(* CODESYS project Flight Simulator Diagnostics.project.export

Project tree, tasks and I/O mapping:
  application Application
    libraries: Unit Conversion Interfaces, * (Intern); Standard, * (System); VisuDialogs, * (System); CAA Device Diagnosis, 3.5.4.0 (CAA Technical Workgroup); CAA Net Base Services, 3.5.8.10 (CAA Technical Workgroup); NetVarUdp, 3.5.17.0 (System); PRO JSON, 1.0.0.13 (Pro Electric)
    task EtherCAT_Task (cyclic, interval 8 ms, priority 1) calls nothing
    task VISU_TASK (cyclic, interval 200 ms, priority 31) calls VisuElems.Visu_Prg
    task Task (cyclic, interval 5 ms, priority 1) calls main, TcpClient
    global variables gvlSetting
    data type ServoData
    program TcpClient [ST]
    program main [ST]
    visualisation Main
    global variables GVL
    program DriveDiagnostics [ST]
    function AppendDiagnosticText [ST]
    function BuildDiagnosticFeedback [ST]
*)

// Application/ServoData
TYPE ServoData :
STRUCT
	positions: ARRAY[1..6] OF JSONVAR;
	speeds: ARRAY[1..6] OF JSONVAR;
END_STRUCT
END_TYPE

// Application/gvlSetting
{attribute 'qualified_only'}
VAR_GLOBAL CONSTANT
    // Port to use to send data.
	gc_uiPort        : UINT := 32760;
    // IP Address of the computer that hosts the software.
	gc_stIpAddr      : NBS.IP_ADDR := (sAddr := '192.168.137.123');
	// Length of the telegram.
    gc_wMaxTelegram  : INT := 512;
END_VAR

// Application/GVL
{attribute 'qualified_only'}
VAR_GLOBAL
	// Red light on electrical housing.
	lightRed: BOOL;
	// Yellow light on electrical housing.
	lightYellow: BOOL;
	// Green light on electrical housing.
	lightGreen: BOOL;
	// Reset button on electrical housing.
	resetButton: BOOL := FALSE;
	// Start button on electrical housing.
	startButton: BOOL := FALSE;
	// Stop button on electrical housing.
	stopButton: BOOL := FALSE;
	// Safety system, connected to safety relay.
	safetySystem: BOOL := FALSE;
	// Virtual reset button on HMI.
	resetHMI: BOOL;
	// Virtual start button on HMI.
	startHMI: BOOL;
	// Virtual stop button on HMI.
	stopHMI: BOOL;
	// Virtual toggle button to toggle between tCP data and manual data on HMI.
	useTCPData: BOOL := TRUE;
	// Manual slider velocity input on HMI.
	nextVelocityInput: REAL := 200;
	// Manual slider position input on HMI.
	nextPositionInput: REAL := 0;
	// Flight simulator object.
	FlightSimulator: FlightSimulator;
	// Velocity input from TCP data or HMI data.
	servoVelocities: ARRAY[1..6] OF REAL;
	// Position input from TCP data or HMI data.
	servoPositions: ARRAY[1..6] OF REAL;
	// Current Positions in array format.
	servoPositionsCurrent: ARRAY[1..6] OF REAL;
	// Current Positions in JSON format, used to send back to TCP client.
	currentPositions: ARRAY[1..6] OF JSONVAR;
END_VAR

// Application/main
PROGRAM main
VAR
	bInit: BOOL := TRUE;
	iCounter : INT;
	bEnabled: BOOL;
	iDataUpdated: INT := 0;
	tonTimer: TON;
	UpdateCount: INT := 0;
END_VAR

IF bInit THEN
	GVL.FlightSimulator.init(
		axis1 := servo_drive_1,
		axis2 := servo_drive_2,
		axis3 := servo_drive_3,
		axis4 := servo_drive_4,
		axis5 := servo_drive_5,
		axis6 := servo_drive_6,
		GVL.lightRed,
		GVL.lightYellow,
		GVL.lightGreen,
		enabled := bEnabled,
		safetySystem := GVL.safetySystem,
		newPositions := GVL.servoPositions,
		newVelocities := GVL.servoVelocities
	);
	bInit := FALSE;
END_IF

// Handle reset buttons.
IF GVL.resetButton OR GVL.resetHMI THEN // blauwe knop
	bEnabled := FALSE;
	GVL.FlightSimulator.doReset();
	
	// [NEW] Reset position data zodat platform niet naar oude waarden springt
	FOR iCounter := 1 TO 6 DO
		GVL.currentPositions[iCounter].Number := 0.0;
		GVL.servoPositions[iCounter] := 0.0;
		GVL.servoVelocities[iCounter] := 0.0;
	END_FOR
END_IF

// Handle start buttons.
IF GVL.startButton OR GVL.startHMI THEN // witte knop
	bEnabled := TRUE;
END_IF

// Handle stop buttons
IF GVL.stopButton OR GVL.stopHMI THEN // zwarte knop
	bEnabled := FALSE;
END_IF

// Go through all positions and velocities.
FOR iCounter := 1 TO 6 BY 1 DO 
	IF GVL.useTCPData THEN
		// Always use latest TCP data (don't wait for parseJSON.Done)
		GVL.servoPositions[iCounter] := tcpClient.servoData.positions[iCounter].Number;
		GVL.servoVelocities[iCounter] := tcpClient.servoData.speeds[iCounter].Number;
		
		// Optional: track successful updates for diagnostics
		IF tcpClient.parseJSON.Done THEN
			UpdateCount := UpdateCount + 1;
		END_IF
	ELSE
		// Else take the data from the sliders from the HMI.
		GVL.servoPositions[iCounter] := GVL.nextPositionInput;
		GVL.servoVelocities[iCounter] := GVL.nextVelocityInput;
	END_IF
END_FOR

//THIS^.signal.green.enable := FALSE;
//THIS^.signal.green.blink := FALSE;
//THIS^.signal.green.enable := FALSE;
//THIS^.signal.green.blink := FALSE;

// Cycle sub functions.
GVL.FlightSimulator.cycle();

// Get current positions, used for TcpClient.
FOR iCounter := 1 TO 6 BY 1 DO
	GVL.currentPositions[iCounter].Number := GVL.FlightSimulator.axis[iCounter].getPosition();
	GVL.servoPositionsCurrent[iCounter] := GVL.FlightSimulator.axis[iCounter].getPosition();
END_FOR

END_PROGRAM

// Application/TcpClient
PROGRAM TcpClient
VAR

    // Client object that connects to client machine.
	fbTcpClient   : NBS.TCP_Client;
    // Read object that reads incomming data from client machine.
	fbTcpRead     : NBS.TCP_Read;
    // Write object that writes data to client machine.
	fbTcpWrite    : NBS.TCP_Write;
	
	// TON object for reset delay.
	tonResetDelay: TON;
	// Received telegram from Read object.
	received      : STRING(gvlSetting.gc_wMaxTelegram);
	// Sent telegram to Write object.
	sent          : STRING(4095);
	// JSON Parser object to parse read data.
	parseJSON     : JSON_TO_STRUCT;
	// JSON Composer object to compose data to write.
	composeJSON   : STRUCT_TO_JSON;
	// Struct that stores the received data in usable arrays.
	servoData     : ServoData;
    // Make connection.
	xConnect      : BOOL := TRUE;
	// Do composing.
	xCompose: BOOL;
	// Do write action.
	xWrite: BOOL;
	// Do parsing
	xParse: BOOL;
	
	j : INT := 1;
 
    // Do read action.
	xRead         : BOOL;
    // Size of read data telegram.
	udiRead       : UDINT;
	// Timeout in µs.
	udiTimeOut: UDINT := 500000;
	
	
	udiVal        : UDINT;
    pudiVal       : POINTER TO BYTE;
    iIndex        : INT;
	xMissingAck   : BOOL;
    udiResult     : UDINT;
    udiLastAck    : UDINT;
    udiNow        : UDINT;
    diagnosticSendTimer : TON;
    diagnosticBuildErrors : UDINT;
END_VAR

 fbTcpClient(xEnable := xConnect, ipAddr := gvlSetting.gc_stIpAddr, uiPort := gvlSetting.gc_uiPort, udiTimeOut := udiTimeOut);
// 
// // Run when connection is active.
// IF fbTcpClient.xActive AND GVL.FlightSimulator.isInitialised() THEN
// 	
// 	IF fbTcpWrite.xDone THEN
// 		xWrite := FALSE;
// 	ELSIF NOT fbTcpWrite.xBusy THEN
// 		IF composeJSON.Done AND composeJSON.Execute THEN
// 			xCompose := FALSE;
// 			xWrite := TRUE;
// 		ELSIF (NOT composeJSON.Busy) THEN
// 			   xCompose := TRUE;
// 			   xWrite := FALSE;
// 		END_IF
// 	END_IF
// 	
// 	composeJSON(
// 		Execute:= xCompose,
// 		JSONString:= ADR(sent),
// 		JSONStringSize:= SIZEOF(sent),
// 		JSONVars:= ADR(GVL.currentPositions),
// 		NumberOfVars:= SIZEOF(GVL.currentPositions) / SIZEOF(JSONVAR)
// 	); 
// 	fbTcpWrite(xExecute := xWrite, hConnection := fbTcpClient.hConnection, udiTimeOut := udiTimeOut, szSize := SIZEOF(sent), pData := ADR(sent));
// 	
// 	IF (NOT fbTcpRead.xBusy) AND (NOT parseJSON.Busy) THEN
// 		xRead := TRUE;
// 	ELSIF fbTcpRead.xReady THEN
// 		xRead := FALSE;
// 		xParse := TRUE;
// 	ELSIF (NOT parseJSON.Busy) THEN
// 		xParse := FALSE;
// 	END_IF
// 
// 	parseJSON(
// 		Execute := xParse,
// 		JSONString:= ADR(received),
// 		JSONStringSize:= SIZEOF(received),
// 		JSONVars:= ADR(servoData),
// 		NumberOfVars:= SIZEOF(servoData) / SIZEOF(JSONVAR)
// 	);
// 	
// 	received := '';
// 	//FOR j := 1 TO SIZEOF(received) DO
// 	//	received[j] := 0;
// 	//END_FOR
// 	//sent := '';
// 	fbTcpRead(xEnable := xRead, hConnection := fbTcpClient.hConnection, szSize := SIZEOF(received), pData := ADR(received), szCount => udiRead);
// 	
// END_IF
// 
// // Reset connection when connection has stopped.
// IF (NOT xConnect) THEN
// 	// Reset all variables.
// 	xConnect := FALSE;
// 	xWrite := FALSE;
// 	xCompose := FALSE;
// 	fbTcpWrite(xExecute := FALSE);
// 	xRead := FALSE;
// 	xParse := FALSE;
// 	fbTcpRead(xEnable := FALSE);
// 	received := '';
// 	sent := '';
// 	// Delay reset for 3 sec.
// 	tonResetDelay(IN:=TRUE, PT:=T#3S);
// 	IF (tonResetDelay.Q) THEN
// 		tonResetDelay(IN:=FALSE);
// 		xConnect := TRUE;
// 	END_IF
// 	
// END_IF
// 
// IF fbTcpClient.xDone AND xConnect THEN
// 	xConnect := FALSE;
// END_IF
// 
// // Stop connection when in error.
// //IF fbTcpClient.xError OR fbTcpWrite.xError OR fbTcpRead.xError THEN
// IF fbTcpClient.xError OR fbTcpRead.xError THEN
// 
// 	xConnect := FALSE;
// 	fbTcpWrite(xExecute := FALSE);
// END_IF 
// 

// Run when connection is active.
IF fbTcpClient.xActive AND GVL.FlightSimulator.isInitialised() THEN
    DriveDiagnostics();
    diagnosticSendTimer(IN := NOT xWrite, PT := T#50MS);
    IF fbTcpWrite.xDone OR fbTcpWrite.xError THEN
        xWrite := FALSE;
    ELSIF NOT fbTcpWrite.xBusy AND diagnosticSendTimer.Q THEN
        sent := BuildDiagnosticFeedback();
        xWrite := LEN(sent) > 0;
        IF NOT xWrite THEN diagnosticBuildErrors := diagnosticBuildErrors + 1; END_IF
    END_IF
    // Buffer remains unchanged while TCP_Write is busy. Send only meaningful
    // bytes (including the newline), never the unused NUL-filled capacity.
    fbTcpWrite(xExecute := xWrite, hConnection := fbTcpClient.hConnection,
        udiTimeOut := udiTimeOut, szSize := INT_TO_UDINT(LEN(sent)), pData := ADR(sent));

    // -------------------------
    //  ONTVANGEN VAN STUARTSERVER
    // -------------------------
    IF (NOT fbTcpRead.xBusy) AND (NOT parseJSON.Busy) THEN
        xRead := TRUE;
    ELSIF fbTcpRead.xReady THEN
        xRead := FALSE;
        xParse := TRUE;
    ELSIF (NOT parseJSON.Busy) THEN
        xParse := FALSE;
    END_IF

    parseJSON(
        Execute         := xParse,
        JSONString      := ADR(received),
        JSONStringSize  := SIZEOF(received),
        JSONVars        := ADR(servoData),
        NumberOfVars    := SIZEOF(servoData) / SIZEOF(JSONVAR)
    );

    // Buffer leegmaken voor volgende receive
    received := '';
    fbTcpRead(
        xEnable    := xRead,
        hConnection:= fbTcpClient.hConnection,
        szSize     := SIZEOF(received),
        pData      := ADR(received),
        szCount    => udiRead
    );

END_IF


// Reset connection when connection has stopped.
 IF (NOT xConnect) THEN
 	// Reset all variables.
 	xConnect := FALSE;
 	xWrite := FALSE;
 	xCompose := FALSE;
	fbTcpWrite(xExecute := FALSE);
 	xRead := FALSE;
 	xParse := FALSE;
 	fbTcpRead(xEnable := FALSE);
	received := '';
 	sent := '';
 	// Delay reset for 3 sec.
 	tonResetDelay(IN:=TRUE, PT:=T#3S);
 	IF (tonResetDelay.Q) THEN
 		tonResetDelay(IN:=FALSE);
 		xConnect := TRUE;
 	END_IF
	
 END_IF
 
 IF fbTcpClient.xDone AND xConnect THEN
 	xConnect := FALSE;
 END_IF

 // Stop connection when in error.
 //IF fbTcpClient.xError OR fbTcpWrite.xError OR fbTcpRead.xError THEN
IF fbTcpClient.xError OR fbTcpRead.xError THEN

	xConnect := FALSE;
	fbTcpWrite(xExecute := FALSE);
END_IF

END_PROGRAM

// Application/DriveDiagnostics
PROGRAM DriveDiagnostics
VAR
    // Passive readers only. No command, enable, reset, or axis configuration writes.
    positionReaders : ARRAY[1..6] OF MC_ReadActualPosition_Festo;
    velocityReaders : ARRAY[1..6] OF MC_ReadActualVelocity_Festo;
    parameterReader : MC_ReadParameter_Festo;
    actualPositions : ARRAY[1..6] OF REAL;
    actualVelocities : ARRAY[1..6] OF REAL;
    positionValid : ARRAY[1..6] OF BOOL;
    velocityValid : ARRAY[1..6] OF BOOL;
    driveTargets : ARRAY[1..6] OF LREAL;
    followingErrors : ARRAY[1..6] OF LREAL;
    targetNew : ARRAY[1..6] OF BOOL;
    followingNew : ARRAY[1..6] OF BOOL;
    targetTick : ARRAY[1..6] OF UDINT;
    followingTick : ARRAY[1..6] OF UDINT;
    readErrors : ARRAY[1..6] OF WORD;
    readErrorCount : UDINT;
    sampleSequence : UDINT;
    sampleTick : UDINT;
    pollAxis : INT := 1;
    pollFollowing : BOOL;
    pollActive : BOOL;
    pollReset : BOOL;
    pollInterval : TON;
    pollTimeout : TON;
    parameter : UINT;
    drive : REFERENCE TO AXIS_REF_FESTO;
    i : INT;
END_VAR

// User units are supplied by the Festo library. Valid AND NOT Error is required;
// never turn a failed read into a plausible zero-valued measurement.
positionReaders[1](Axis := servo_drive_1, Enable := TRUE);
positionReaders[2](Axis := servo_drive_2, Enable := TRUE);
positionReaders[3](Axis := servo_drive_3, Enable := TRUE);
positionReaders[4](Axis := servo_drive_4, Enable := TRUE);
positionReaders[5](Axis := servo_drive_5, Enable := TRUE);
positionReaders[6](Axis := servo_drive_6, Enable := TRUE);
velocityReaders[1](Axis := servo_drive_1, Enable := TRUE);
velocityReaders[2](Axis := servo_drive_2, Enable := TRUE);
velocityReaders[3](Axis := servo_drive_3, Enable := TRUE);
velocityReaders[4](Axis := servo_drive_4, Enable := TRUE);
velocityReaders[5](Axis := servo_drive_5, Enable := TRUE);
velocityReaders[6](Axis := servo_drive_6, Enable := TRUE);
sampleTick := TIME_TO_UDINT(TIME());
FOR i := 1 TO 6 DO
    positionValid[i] := positionReaders[i].Valid AND NOT positionReaders[i].Error;
    velocityValid[i] := velocityReaders[i].Valid AND NOT velocityReaders[i].Error;
    actualPositions[i] := positionReaders[i].Position;
    actualVelocities[i] := velocityReaders[i].Velocity;
END_FOR

// Only one SDO request is active across all six drives. Each request is followed
// by a 50 ms idle interval. Register traces are slower than the 20 Hz PDO traces.
// Do not increase this rate without measuring the actual fieldbus load.
CASE pollAxis OF
    1: drive REF= servo_drive_1;
    2: drive REF= servo_drive_2;
    3: drive REF= servo_drive_3;
    4: drive REF= servo_drive_4;
    5: drive REF= servo_drive_5;
    6: drive REF= servo_drive_6;
END_CASE
IF pollFollowing THEN parameter := 16#60F4; ELSE parameter := 16#607A; END_IF
IF pollReset THEN
    parameterReader(Axis := drive, Enable := FALSE);
    pollTimeout(IN := FALSE);
    pollInterval(IN := FALSE);
    pollReset := FALSE;
    IF pollFollowing THEN
        pollAxis := pollAxis + 1;
        IF pollAxis > 6 THEN pollAxis := 1; END_IF
    END_IF
    pollFollowing := NOT pollFollowing;
ELSE
    pollInterval(IN := NOT pollActive, PT := T#50MS);
    IF pollInterval.Q THEN pollActive := TRUE; END_IF
    parameterReader(Axis := drive, Enable := pollActive,
        ParameterNumber := parameter, SubindexNumber := 0);
    pollTimeout(IN := pollActive, PT := T#1S);
    IF pollActive AND (parameterReader.Valid OR parameterReader.Error OR pollTimeout.Q) THEN
        IF parameterReader.Valid AND NOT parameterReader.Error THEN
            IF pollFollowing THEN
                followingErrors[pollAxis] := parameterReader.Value;
                followingTick[pollAxis] := sampleTick;
                followingNew[pollAxis] := TRUE;
            ELSE
                driveTargets[pollAxis] := parameterReader.Value;
                targetTick[pollAxis] := sampleTick;
                targetNew[pollAxis] := TRUE;
            END_IF
            readErrors[pollAxis] := 0;
        ELSE
            readErrorCount := readErrorCount + 1;
            IF pollTimeout.Q THEN readErrors[pollAxis] := 16#FFFF;
            ELSE readErrors[pollAxis] := parameterReader.ErrorID; END_IF
            IF pollFollowing THEN followingNew[pollAxis] := FALSE;
            ELSE targetNew[pollAxis] := FALSE; END_IF
        END_IF
        pollActive := FALSE;
        pollReset := TRUE;
    END_IF
END_IF

END_PROGRAM

// Application/BuildDiagnosticFeedback
FUNCTION BuildDiagnosticFeedback : STRING(4095)
VAR
    output : STRING(4095);
    fragment : STRING(255);
    field : INT;
    i : INT;
    valid : BOOL;
    ok : BOOL := TRUE;
END_VAR

output := '{"currentPositions":[';
ok := TRUE;
FOR i := 1 TO 6 DO
    IF i > 1 THEN ok := AppendDiagnosticText(',', output) AND ok; END_IF
    ok := AppendDiagnosticText(REAL_TO_STRING(GVL.currentPositions[i].Number), output) AND ok;
END_FOR
ok := AppendDiagnosticText('],"diagnostics":{"version":1,"sequence":', output) AND ok;
DriveDiagnostics.sampleSequence := DriveDiagnostics.sampleSequence + 1;
ok := AppendDiagnosticText(UDINT_TO_STRING(DriveDiagnostics.sampleSequence), output) AND ok;
ok := AppendDiagnosticText(',"plcTickMs":', output) AND ok;
ok := AppendDiagnosticText(UDINT_TO_STRING(DriveDiagnostics.sampleTick), output) AND ok;
ok := AppendDiagnosticText(',"sdoReadErrors":', output) AND ok;
ok := AppendDiagnosticText(UDINT_TO_STRING(DriveDiagnostics.readErrorCount), output) AND ok;
ok := AppendDiagnosticText(',"positionUnit":"Festo user unit","velocityUnit":"Festo user unit/s","registerUnit":"raw CiA402","followingErrorSource":"0x60F4 readback","targetSource":"0x607A readback"', output) AND ok;
// Field order is fixed; actuator order stays A1..A6. Null means no new valid
// sample. SDO sample ticks are kept separately from packet assembly time.
FOR field := 1 TO 11 DO
    CASE field OF
        1: fragment := ',"receivedPositions":[';
        2: fragment := ',"receivedSpeeds":[';
        3: fragment := ',"actualPositions":[';
        4: fragment := ',"actualVelocities":[';
        5: fragment := ',"driveTargetPositions":[';
        6: fragment := ',"followingErrors":[';
        7: fragment := ',"targetSampleTickMs":[';
        8: fragment := ',"followingSampleTickMs":[';
        9: fragment := ',"sdoErrorIds":[';
        10: fragment := ',"requestedPositions":[';
        11: fragment := ',"requestedSpeeds":[';
    END_CASE
    ok := AppendDiagnosticText(fragment, output) AND ok;
    FOR i := 1 TO 6 DO
        IF i > 1 THEN ok := AppendDiagnosticText(',', output) AND ok; END_IF
        valid := TRUE;
        CASE field OF
            1: fragment := REAL_TO_STRING(TcpClient.servoData.positions[i].Number);
            2: fragment := REAL_TO_STRING(TcpClient.servoData.speeds[i].Number);
            3: fragment := REAL_TO_STRING(DriveDiagnostics.actualPositions[i]); valid := DriveDiagnostics.positionValid[i];
            4: fragment := REAL_TO_STRING(DriveDiagnostics.actualVelocities[i]); valid := DriveDiagnostics.velocityValid[i];
            5: fragment := LREAL_TO_STRING(DriveDiagnostics.driveTargets[i]); valid := DriveDiagnostics.targetNew[i];
            6: fragment := LREAL_TO_STRING(DriveDiagnostics.followingErrors[i]); valid := DriveDiagnostics.followingNew[i];
            7: fragment := UDINT_TO_STRING(DriveDiagnostics.targetTick[i]); valid := DriveDiagnostics.targetNew[i];
            8: fragment := UDINT_TO_STRING(DriveDiagnostics.followingTick[i]); valid := DriveDiagnostics.followingNew[i];
            9: fragment := UINT_TO_STRING(WORD_TO_UINT(DriveDiagnostics.readErrors[i]));
            10: fragment := REAL_TO_STRING(GVL.servoPositions[i]);
            11: fragment := REAL_TO_STRING(GVL.servoVelocities[i]);
        END_CASE
        IF NOT valid THEN fragment := 'null'; END_IF
        ok := AppendDiagnosticText(fragment, output) AND ok;
    END_FOR
    ok := AppendDiagnosticText(']', output) AND ok;
END_FOR
ok := AppendDiagnosticText('}}$N', output) AND ok;
IF ok THEN
    BuildDiagnosticFeedback := output;
    FOR i := 1 TO 6 DO
        DriveDiagnostics.targetNew[i] := FALSE;
        DriveDiagnostics.followingNew[i] := FALSE;
    END_FOR
ELSE
    // Never send truncated JSON. TcpClient counts this failure for inspection.
    BuildDiagnosticFeedback := '';
END_IF

END_FUNCTION

// Application/AppendDiagnosticText
FUNCTION AppendDiagnosticText : BOOL
VAR_INPUT
    fragment : STRING(255);
END_VAR
VAR_IN_OUT
    destination : STRING(4095);
END_VAR
VAR
    used : INT;
    count : INT;
    i : INT;
    outputBytes : POINTER TO BYTE;
    inputBytes : POINTER TO BYTE;
END_VAR

// Standard CONCAT may return STRING(255). Explicit bounded copying preserves
// larger feedback objects and always leaves a terminating NUL in PLC memory.
used := LEN(destination);
count := LEN(fragment);
AppendDiagnosticText := used + count <= 4095;
IF NOT AppendDiagnosticText THEN RETURN; END_IF
outputBytes := ADR(destination);
inputBytes := ADR(fragment);
FOR i := 0 TO count - 1 DO outputBytes[used + i] := inputBytes[i]; END_FOR
outputBytes[used + count] := 0;

END_FUNCTION

// Application/Main
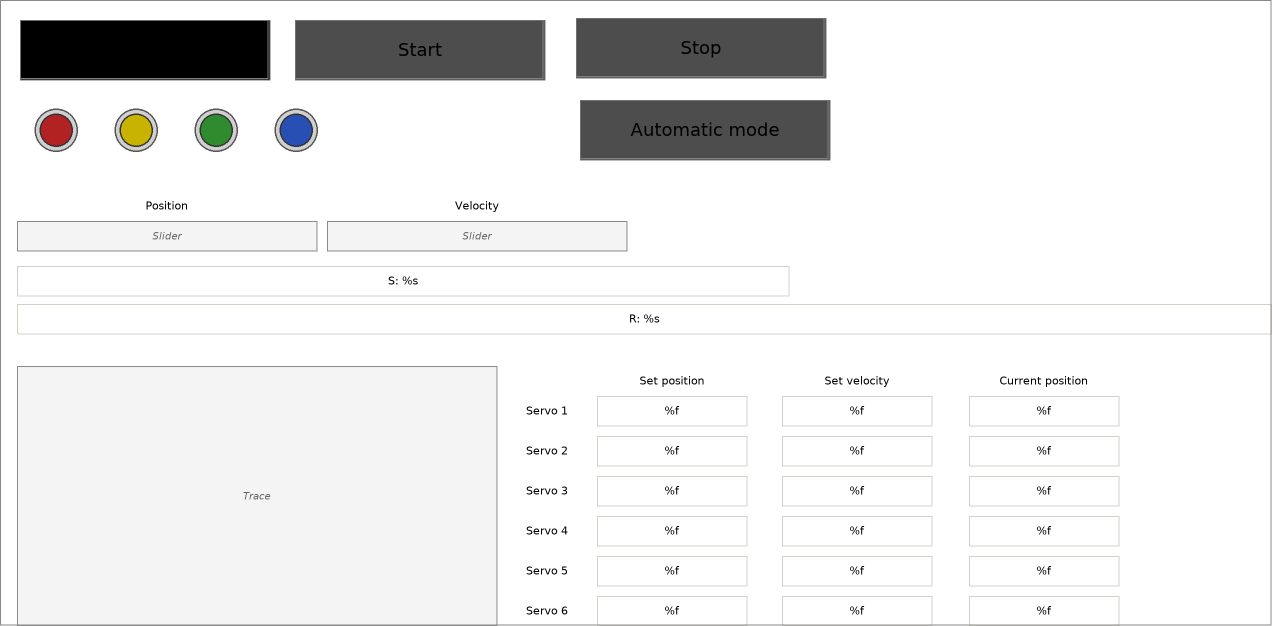
VISUALIZATION Main  // 1272x626
    Button (20,20 250x60), "Reset"
        tap GVL.resetHMI
    Button (295,20 250x60), "Start"
        tap GVL.startHMI
    Slider (17,221 300x30), scale 10..390
    Button (580,100 250x60), "Automatic mode"
        toggle GVL.usetcpdata
    Slider (327,221 300x30), scale 0..400
    Button (576,18 250x60), "Stop"
        tap GVL.stopHMI
    Lamp1 (191,105 50x50), variable: GVL.lightGreen, style: Lamp-Lamp1-Green
    Lamp1 (31,105 50x50), variable: GVL.lightRed, style: Lamp-Lamp1-Red
    Lamp1 (111,105 50x50), variable: GVL.lightYellow, style: Lamp-Lamp1-Yellow
    Textfield (17,266 772x30), "S: %s", text variable: TcpClient.sent
    Textfield (17,304 1255x30), "R: %s", text variable: TcpClient.received
    Textfield (597,396 150x30), "%f", text variable: GVL.servoPositions[1]
        OnMouseClick: write the text variable via InputWithLimits, min 0, max 400
    Textfield (597,436 150x30), "%f", text variable: GVL.servoPositions[2]
        OnMouseClick: write the text variable via InputWithLimits, min 0, max 400
    Textfield (597,476 150x30), "%f", text variable: GVL.servoPositions[3]
        OnMouseClick: write the text variable via InputWithLimits, min 0, max 400
    Textfield (597,516 150x30), "%f", text variable: GVL.servoPositions[4]
        OnMouseClick: write the text variable via InputWithLimits, min 0, max 400
    Textfield (597,556 150x30), "%f", text variable: GVL.servoPositions[5]
        OnMouseClick: write the text variable via InputWithLimits, min 0, max 400
    Textfield (597,596 150x30), "%f", text variable: GVL.servoPositions[6]
        OnMouseClick: write the text variable via InputWithLimits, min 0, max 400
    Textfield (782,396 150x30), "%f", text variable: GVL.servoVelocities[1]
        OnMouseClick: write the text variable via InputWithLimits, min 0, max 400
    Textfield (782,436 150x30), "%f", text variable: GVL.servoVelocities[2]
        OnMouseClick: write the text variable via InputWithLimits, min 0, max 400
    Textfield (782,476 150x30), "%f", text variable: GVL.servoVelocities[3]
        OnMouseClick: write the text variable via InputWithLimits, min 0, max 400
    Textfield (782,516 150x30), "%f", text variable: GVL.servoVelocities[4]
        OnMouseClick: write the text variable via InputWithLimits, min 0, max 400
    Textfield (782,556 150x30), "%f", text variable: GVL.servoVelocities[5]
        OnMouseClick: write the text variable via InputWithLimits, min 0, max 400
    Textfield (782,596 150x30), "%f", text variable: GVL.servoVelocities[6]
        OnMouseClick: write the text variable via InputWithLimits, min 0, max 400
    Label (597,366 150x30), "Set position"
    Label (782,366 150x30), "Set velocity"
    Label (497,396 100x30), "Servo 1"
    Label (497,436 100x30), "Servo 2"
    Label (497,476 100x30), "Servo 3"
    Label (497,516 100x30), "Servo 4"
    Label (497,556 100x30), "Servo 5"
    Label (497,596 100x30), "Servo 6"
    Lamp1 (271,105 50x50), variable: GVL.FlightSimulator.isReady(), style: Lamp-Lamp1-Blue
    Trace (17,366 480x260)
    Textfield (969,396 150x30), "%f", text variable: GVL.servoPositionsCurrent[1]
        OnMouseClick: write the text variable via InputWithLimits, min 0, max 400
    Textfield (969,436 150x30), "%f", text variable: GVL.servoPositionsCurrent[2]
        OnMouseClick: write the text variable via InputWithLimits, min 0, max 400
    Textfield (969,476 150x30), "%f", text variable: GVL.servoPositionsCurrent[3]
        OnMouseClick: write the text variable via InputWithLimits, min 0, max 400
    Textfield (969,516 150x30), "%f", text variable: GVL.servoPositionsCurrent[4]
        OnMouseClick: write the text variable via InputWithLimits, min 0, max 400
    Textfield (969,556 150x30), "%f", text variable: GVL.servoPositionsCurrent[5]
        OnMouseClick: write the text variable via InputWithLimits, min 0, max 400
    Textfield (969,596 150x30), "%f", text variable: GVL.servoPositionsCurrent[6]
        OnMouseClick: write the text variable via InputWithLimits, min 0, max 400
    Label (969,366 150x30), "Current position"
    Label (92,191 150x30), "Position"
    Label (402,191 150x30), "Velocity"
END_VISUALIZATION
